FUNCTION ENCODERtoANGLE : REAL
VAR_INPUT
	encoder_in : UDINT;
	
END_VAR
VAR
	Pulsos : UDINT :=600;
END_VAR

///Medir ángulos
ENCODERtoANGLE:= 2*GVL.Pi - (encoder_in MOD Pulsos)*2*GVL.Pi/Pulsos;

END_FUNCTION

(* stored: Version 1.1.0.1, ProductVersion 3.1.4024.4
   POU ENCODERtoANGLE: Id {0b3edcd1-9b78-46ac-a2a6-6cfa1826f812}, SpecialFunc None *)
